FUNCTION_BLOCK FB_DigitalSensNO
VAR_INPUT
	_input	: BOOL;
END_VAR

VAR_OUTPUT
	_output : BOOL;
END_VAR

_output := _input;

PROPERTY IsActive : BOOL
GET
IsActive:= _output;
END_GET
END_PROPERTY

END_FUNCTION_BLOCK

(* stored: Version 1.1.0.1, ProductVersion 3.1.4024.16
   POU FB_DigitalSensNO: Id {9b7f398c-5bf7-4085-9c37-3cc19cb2758d}, SpecialFunc None
   Property IsActive: Id {d21f2347-78c6-48ff-b8b4-4796ac7e56b7}
   Get Get: Id {10566830-eb48-451a-8cea-d902e630293f} *)
